LIN {X 0,Y 137.056,Z 476.203,A -85,B 0,C 180,E1 -30599.195,E2 -30599.195} C_VEL
LIN {X 0,Y 140.564,Z 471.572,A -85,B 0,C 180,E1 -30599.428,E2 -30599.428} C_VEL
LIN {X 0,Y 140.56,Z 471.582,A -85,B 0,C 180,E1 -30599.574,E2 -30599.574} C_VEL
LIN {X 0,Y 130.958,Z 483.52,A -85,B 0,C 180,E1 -30600.213,E2 -30600.213} C_VEL
LIN {X 0,Y 121.245,Z 493.76,A -85,B 0,C 180,E1 -30600.887,E2 -30600.887} C_VEL
LIN {X 0,Y 110.739,Z 503.148,A -85,B 0,C 180,E1 -30601.729,E2 -30601.729} C_VEL
LIN {X 0,Y 98.529,Z 512.388,A -85,B 0,C 180,E1 -30603.046,E2 -30603.046} C_VEL
LIN {X 0,Y 87.189,Z 519.608,A -85,B 0,C 180,E1 -30604.623,E2 -30604.623} C_VEL
LIN {X 0,Y 74.379,Z 526.468,A -85,B 0,C 180,E1 -30607.203,E2 -30607.203} C_VEL
LIN {X 0,Y 60.839,Z 532.345,A -85,B 0,C 180,E1 -30610.925,E2 -30610.925} C_VEL
LIN {X 0,Y 50.938,Z 535.849,A -85,B 0,C 180,E1 -30615.032,E2 -30615.032} C_VEL
LIN {X 0,Y 38.363,Z 539.396,A -85,B 0,C 180,E1 -30623.656,E2 -30623.656} C_VEL
LIN {X 0,Y 27.347,Z 541.74,A -85,B 0,C 180,E1 -30639.559,E2 -30639.559} C_VEL
LIN {X 0,Y 20.52,Z 542.937,A -85,B 0,C 180,E1 -30669.972,E2 -30669.972} C_VEL
LIN {X 0,Y 19.928,Z 543.104,A -85,B 0,C 180,E1 -30690,E2 -30690} C_VEL
LIN {X 0,Y 23.144,Z 542.456,A -85,B 0,C 180,E1 -30727.396,E2 -30727.396} C_VEL
LIN {X 0,Y 32.553,Z 540.657,A -85,B 0,C 180,E1 -30749.719,E2 -30749.719} C_VEL
LIN {X 0,Y 45.536,Z 537.393,A -85,B 0,C 180,E1 -30762.021,E2 -30762.021} C_VEL
LIN {X 0,Y 57.504,Z 533.49,A -85,B 0,C 180,E1 -30767.881,E2 -30767.881} C_VEL
LIN {X 0,Y 70.966,Z 527.944,A -85,B 0,C 180,E1 -30772.018,E2 -30772.018} C_VEL
LIN {X 0,Y 84.669,Z 520.901,A -85,B 0,C 180,E1 -30774.898,E2 -30774.898} C_VEL
LIN {X 0,Y 96.788,Z 513.379,A -85,B 0,C 180,E1 -30776.758,E2 -30776.758} C_VEL
LIN {X 0,Y 108.992,Z 504.323,A -85,B 0,C 180,E1 -30778.089,E2 -30778.089} C_VEL
LIN {X 0,Y 119.492,Z 495.082,A -85,B 0,C 180,E1 -30778.997,E2 -30778.997} C_VEL
LIN {X 0,Y 129.687,Z 484.565,A -85,B 0,C 180,E1 -30779.717,E2 -30779.717} C_VEL
LIN {X 0,Y 139.681,Z 472.316,A -85,B 0,C 180,E1 -30780.391,E2 -30780.391} C_VEL
LIN {X 0,Y 140.561,Z 471.139,A -85,B 0,C 180,E1 -30780.436,E2 -30780.436} C_VEL
LIN {X 0,Y 140.566,Z 471.124,A -85,B 0,C 180,E1 -30780.648,E2 -30780.648} C_VEL
LIN {X 0,Y 140.604,Z 473.124,A -85,B 0,C 180,E1 -30781.486,E2 -30781.486} C_VEL
LIN {X 0,Y 140.604,Z 526.4,A -85,B 0,C 180,E1 -30781.486,E2 -30781.486} C_VEL
LIN {X 0,Y 96.407,Z 526.4,A -85,B 0,C 180,E1 -30781.136,E2 -30781.136} C_VEL
LIN {X 0,Y 94.407,Z 524.4,A -85,B 0,C 180,E1 -30781.112,E2 -30781.112} C_VEL
LIN {X 0,Y 94.407,Z 518.217,A -85,B 0,C 180,E1 -30781.112,E2 -30781.112} C_VEL
LIN {X 0,Y 91.388,Z 516.513,A -85,B 0,C 180,E1 -30781.365,E2 -30781.365} C_VEL
LIN {X 0,Y 80.902,Z 522.46,A -85,B 0,C 180,E1 -30782.573,E2 -30782.573} C_VEL
LIN {X 0,Y 67.002,Z 528.997,A -85,B 0,C 180,E1 -30784.821,E2 -30784.821} C_VEL
LIN {X 0,Y 53.256,Z 534.096,A -85,B 0,C 180,E1 -30788.222,E2 -30788.222} C_VEL
LIN {X 0,Y 43.125,Z 537.029,A -85,B 0,C 180,E1 -30792.098,E2 -30792.098} C_VEL
LIN {X 0,Y 30.097,Z 539.887,A -85,B 0,C 180,E1 -30800.931,E2 -30800.931} C_VEL
LIN {X 0,Y 18.645,Z 541.588,A -85,B 0,C 180,E1 -30821.076,E2 -30821.076} C_VEL
LIN {X 0,Y 13.054,Z 542.171,A -85,B 0,C 180,E1 -30870,E2 -30870} C_VEL
LIN {X 0,Y 18.638,Z 541.615,A -85,B 0,C 180,E1 -30918.949,E2 -30918.949} C_VEL
LIN {X 0,Y 30.071,Z 539.949,A -85,B 0,C 180,E1 -30939.2,E2 -30939.2} C_VEL
LIN {X 0,Y 43.12,Z 537.119,A -85,B 0,C 180,E1 -30947.929,E2 -30947.929} C_VEL
LIN {X 0,Y 57.013,Z 532.938,A -85,B 0,C 180,E1 -30952.918,E2 -30952.918} C_VEL
LIN {X 0,Y 70.462,Z 527.674,A -85,B 0,C 180,E1 -30955.859,E2 -30955.859} C_VEL
LIN {X 0,Y 84.385,Z 520.803,A -85,B 0,C 180,E1 -30957.999,E2 -30957.999} C_VEL
LIN {X 0,Y 91.384,Z 516.738,A -85,B 0,C 180,E1 -30958.726,E2 -30958.726} C_VEL
LIN {X 0,Y 91.365,Z 516.773,A -85,B 0,C 180,E1 -30959.507,E2 -30959.507} C_VEL
LIN {X 0,Y 77.321,Z 524.593,A -85,B 0,C 180,E1 -30961.141,E2 -30961.141} C_VEL
LIN {X 0,Y 63.363,Z 530.82,A -85,B 0,C 180,E1 -30963.417,E2 -30963.417} C_VEL
LIN {X 0,Y 49.563,Z 535.647,A -85,B 0,C 180,E1 -30966.987,E2 -30966.987} C_VEL
LIN {X 0,Y 36.089,Z 539.193,A -85,B 0,C 180,E1 -30973.175,E2 -30973.175} C_VEL
LIN {X 0,Y 23.443,Z 541.538,A -85,B 0,C 180,E1 -30985.927,E2 -30985.927} C_VEL
LIN {X 0,Y 14.022,Z 542.735,A -85,B 0,C 180,E1 -31019.92,E2 -31019.92} C_VEL
LIN {X 0,Y 12.817,Z 542.903,A -85,B 0,C 180,E1 -31050,E2 -31050} C_VEL
LIN {X 0,Y 17.996,Z 542.253,A -85,B 0,C 180,E1 -31101.356,E2 -31101.356} C_VEL
LIN {X 0,Y 29.596,Z 540.454,A -85,B 0,C 180,E1 -31121.776,E2 -31121.776} C_VEL
LIN {X 0,Y 42.924,Z 537.44,A -85,B 0,C 180,E1 -31130.577,E2 -31130.577} C_VEL
LIN {X 0,Y 56.437,Z 533.286,A -85,B 0,C 180,E1 -31135.005,E2 -31135.005} C_VEL
LIN {X 0,Y 70.33,Z 527.74,A -85,B 0,C 180,E1 -31137.802,E2 -31137.802} C_VEL
LIN {X 0,Y 84.335,Z 520.695,A -85,B 0,C 180,E1 -31139.787,E2 -31139.787} C_VEL
LIN {X 0,Y 91.366,Z 516.55,A -85,B 0,C 180,E1 -31140.545,E2 -31140.545} C_VEL
LIN {X 0,Y 91.388,Z 516.513,A -85,B 0,C 180,E1 -31141.365,E2 -31141.365} C_VEL
LIN {X 0,Y 91.46,Z 518.512,A -85,B 0,C 180,E1 -31142.654,E2 -31142.654} C_VEL
LIN {X 0,Y 91.46,Z 545.366,A -85,B 0,C 180,E1 -31142.654,E2 -31142.654} C_VEL
LIN {X 0,Y 52.659,Z 545.366,A -85,B 0,C 180,E1 -31140.888,E2 -31140.888} C_VEL
LIN {X 0,Y 50.664,Z 543.366,A -85,B 0,C 180,E1 -31140.724,E2 -31140.724} C_VEL
LIN {X 0,Y 50.664,Z 537.589,A -85,B 0,C 180,E1 -31140.724,E2 -31140.724} C_VEL
LIN {X 0,Y 48.196,Z 535.653,A -85,B 0,C 180,E1 -31141.202,E2 -31141.202} C_VEL
LIN {X 0,Y 35.247,Z 538.809,A -85,B 0,C 180,E1 -31144.472,E2 -31144.472} C_VEL
LIN {X 0,Y 21.544,Z 541.08,A -85,B 0,C 180,E1 -31151.863,E2 -31151.863} C_VEL
LIN {X 0,Y 9.027,Z 542.223,A -85,B 0,C 180,E1 -31178.874,E2 -31178.874} C_VEL
LIN {X 0,Y 5.959,Z 542.372,A -85,B 0,C 180,E1 -31229.999,E2 -31229.999} C_VEL
LIN {X 0,Y 14.957,Z 541.816,A -85,B 0,C 180,E1 -31300.01,E2 -31300.01} C_VEL
LIN {X 0,Y 28.333,Z 540.151,A -85,B 0,C 180,E1 -31312.829,E2 -31312.829} C_VEL
LIN {X 0,Y 42.209,Z 537.32,A -85,B 0,C 180,E1 -31317.427,E2 -31317.427} C_VEL
LIN {X 0,Y 48.033,Z 535.805,A -85,B 0,C 180,E1 -31318.846,E2 -31318.846} C_VEL
LIN {X 0,Y 35.155,Z 538.991,A -85,B 0,C 180,E1 -31321.732,E2 -31321.732} C_VEL
LIN {X 0,Y 21.309,Z 541.335,A -85,B 0,C 180,E1 -31328.339,E2 -31328.339} C_VEL
LIN {X 0,Y 8.625,Z 542.533,A -85,B 0,C 180,E1 -31355.43,E2 -31355.43} C_VEL
LIN {X 0,Y 5.697,Z 542.701,A -85,B 0,C 180,E1 -31410.001,E2 -31410.001} C_VEL
LIN {X 0,Y 14.635,Z 542.051,A -85,B 0,C 180,E1 -31483.826,E2 -31483.826} C_VEL
LIN {X 0,Y 28.189,Z 540.251,A -85,B 0,C 180,E1 -31495.759,E2 -31495.759} C_VEL
LIN {X 0,Y 42.167,Z 537.282,A -85,B 0,C 180,E1 -31500.148,E2 -31500.148} C_VEL
LIN {X 0,Y 48.196,Z 535.653,A -85,B 0,C 180,E1 -31501.202,E2 -31501.202} C_VEL
LIN {X 0,Y 50.694,Z 537.585,A -85,B 0,C 180,E1 -31501.564,E2 -31501.564} C_VEL
LIN {X 0,Y 50.694,Z 600,A -85,B 0,C 180,E1 -31501.564,E2 -31501.564} C_VEL
LIN {X 0,Y 50.694,Z 600,A -85,B 0,C 180,E1 -31501.564,E2 -31501.564}

QRS_NEXT_CUT()

QRS_NEXT()
QRS_HOME()

END
